INTERFACE IPart EXTENDS __SYSTEM.IQueryInterface

PROPERTY id : String(23)
GET
END_GET
SET
END_SET
END_PROPERTY

END_INTERFACE

(* stored: Version 1.1.0.1
   Itf IPart: Id {2cbcf229-0419-419d-b31c-9dcb81b4e994}
   Property id: Id {cf3398aa-f18a-402c-9af0-f471b85f6039}
   Get Get: Id {28397749-f62a-4021-98e4-8d0c34db1554}
   Set Set: Id {6ed364ee-3129-468d-a029-253e6c93c6cb} *)
